Staubli VAL3: advance.dtx

num nIndex
num nIndexExport
num nIndexImport
num nIndexPreset
num nKey
public num nPage
num nRefresh
num nTime = 1
num nView
num nViewExport
num nViewImport
string sEventExport
string sEventImport
string sExport
string sImport
public string sItems
string sMenu
string sMessage
string sMenu8[8]
bool bButton[8]
frame fFrame = {fatherId=world[0]}
